DATA_BLOCK "DB_MyDbFromUdt"
NON_RETAIN

"U_Status"

BEGIN

critical := false;

END_DATA_BLOCK